SUBAPPLICATION logiBUS_AI_Calibrate_3P_IDA_OPC (* logiBUS_AI_IDA (Analog-Eingang) mit 3-Punkt-Kalibrierung (AR_CALIBRATE_3P_REF, unabhaengig gespeicherte Rohwerte X_MIN/X_MID/X_MAX + Referenzwerte MIN_REF/MID_REF/MAX_REF alle INI-persistiert) auf VT-Zahlenfelder (Rohwert + kalibrierter Wert, je eigene CNumberVariable) + Bargraph (kalibriert) + 3 VT-Tasten (C_MIN/C_MID/C_MAX) + OPC-UA (Rohwert DWORD + kalibrierter Wert REAL, generisch, ein Kanal). Fuer Sensoren mit definierter Mittelstellung (z.B. Lenkwinkelsensor: links/geradeaus/rechts) statt reiner 2-Punkt-Linearisierung. *)
  (* Standard: 61499-2; Description: Copyright (c) 2026 Meisterschulen am Ostbahnhof This program and the accompanying materials are made available under the terms of the Eclipse Public License 2.0 which is available at https://www.eclipse.org/legal/epl-2.0/ SPDX-License-Identifier: EPL-2.0 *)
  (* Version 1.2, 2026-09-18, Franz Höpfinger, Meisterschulen am Ostbahnhof, AR_CALIBRATE_3P_REF.C_MIN/C_MID/C_MAX von AX-Sockets auf reine EventInputs umgestellt (Franz-Entscheidung, siehe AR_CALIBRATE_2P_REF) - AX_BOOL_TO_X_MIN/_MID/_MAX entfallen ersatzlos, die Merge-Ketten verbinden jetzt direkt per EventConnection mit CALIBRATE.C_MIN/C_MID/C_MAX. *)
  (* Version 1.3, 2026-09-18, Franz Höpfinger, Meisterschulen am Ostbahnhof, C_MIN/C_MAX-Merge-Ketten (2x E_MERGE_2 in Reihe) durch je einen E_MERGE_3 ersetzt, C_MID-Kette (3x E_MERGE_2) durch einen E_MERGE_4 - OR-Merge ist assoziativ, funktional identisch. Siehe logiBUS_AI_Calibrate_IDA_OPC v1.4. *)
  (* Version 1.4, 2026-09-18, Franz Höpfinger, Meisterschulen am Ostbahnhof, Franz: 'kann eine SUB sein' - logiBUS_AI_IDA+AD_SPLIT_2+AD_PUBLISH_RAW+AD_TO_AUDI+AUDI_SPLIT_2+Q_NumericValue_RAW+AUDI_TO_AR durch neue SubApp logiBUS_AI_Raw_VT_AR_OPC ersetzt, AR_SPLIT_2+AR_PUBLISH_CAL+Q_NumericValue_CAL durch die bereits bestehende SubApp AR_TO_Q_Publish_OPC (dort um optionales INITO ergaenzt) - identisch zu logiBUS_AI_Calibrate_IDA_OPC v1.6. Die AX_SUBSCRIBE_MIN-Init-Kette haengt jetzt an PublishCal.INITO statt AR_PUBLISH_CAL.INITO; die vorherige Verkettung AD_PUBLISH_RAW.INITO->AR_PUBLISH_CAL.INIT entfaellt (beide Publishes sind voneinander unabhaengig, initialisieren jetzt unabhaengig/auto). *)
  (* Version 1.5, 2026-09-18, Franz Höpfinger, Meisterschulen am Ostbahnhof, Franz: 'genau so umbauen wie den anderen' (logiBUS_AI_Calibrate_IDA_OPC) - NUR fuer C_MIN/C_MAX: AX_SUBSCRIBE_MIN/MAX + AX_RF_TRIG_MIN/MAX (Toggle-Subscribe, ID_MIN_READ/ID_MAX_READ, beide ueberall unbenutzt) ersatzlos entfernt, ersetzt durch je eine Button_Method_IE (TriggerMIN/TriggerMAX) mit neuer Methodenadresse ID_MIN_METHOD/ID_MAX_METHOD. C_MID BEWUSST NICHT umgestellt: Fahrwerk_Mittelpunkt_Automatik.SUB (Achslenkung, STG1) triggert C_MID lokal (selbe Station!) ueber genau diesen Toggle-Kanal (ID_MID_READ), weil lokaler CALL_METHOD auf derselben Station laut 4diac-Doku nicht funktioniert (FORTE-Log: 'Cannot perform action CALL_METHOD locally') - siehe Fahrwerk_Mittelpunkt_Automatik.SUB v2.2/BERICHT_2026-09-16 Abschnitt 13-15. AX_SUBSCRIBE_MID/AX_RF_TRIG_MID/SERVER_MID_TRIGGER/E_MERGE_MID (E_MERGE_4) bleiben daher unveraendert bestehen. Die OPC_UA_VERNETZUNG.md Punkt 14-Regel (kein Event-Pegel-Event-Umweg) gilt nur fuer echte CROSS-STATION-Trigger, nicht fuer diesen Sonderfall auf derselben Station. *)
  (* Version 1.6, 2026-09-18, Franz Höpfinger, Meisterschulen am Ostbahnhof, Franz: 'TriggerMIN TriggerMAX bitte TriggerMID genau gleich machen' - Button_C_MID + SERVER_MID_TRIGGER (Button/Methode-Teil) durch eine SubApp TriggerMID (Button_Method_IE) ersetzt, strukturell identisch zu TriggerMIN/TriggerMAX. Der lokale Toggle-Kanal (AX_SUBSCRIBE_MID+AX_RF_TRIG_MID) bleibt bestehen (siehe v1.5-Begruendung), wird aber jetzt sauber getrennt als zusaetzliche Quelle in E_MERGE_MID gemergt (E_MERGE_4 -> E_MERGE_3: TriggerMID.IND + AX_RF_TRIG_MID.ER/EF) statt als 4. Quelle in einem grossen Merge mit SERVER_0 direkt inline verdrahtet zu sein. *)
  (* Version 1.7, 2026-09-18, Franz Höpfinger, Meisterschulen am Ostbahnhof, Franz: 'MID, MIN und MAX sind GLEICH' - AX_SUBSCRIBE_MID/AX_RF_TRIG_MID/E_MERGE_MID (der lokale Toggle-Kanal aus v1.5/v1.6) ersatzlos entfernt, ID_MID_READ entfaellt. TriggerMID ist jetzt eine reine Button_Method_IE-Instanz, 1:1 baugleich zu TriggerMIN/TriggerMAX, direkt auf CALIBRATE.C_MID verdrahtet. ACHTUNG: Fahrwerk_Mittelpunkt_Automatik.SUB (Achslenkung/Hangausgleich) toggelt/publiziert weiterhin auf den bisherigen ID_MID_TRIGGER_WRITE-Knoten, den jetzt niemand mehr abonniert - dieser Pfad ist damit funktionslos, bis Fahrwerk_Mittelpunkt_Automatik.SUB auf einen Aufruf von ID_MID_TRIGGER_METHOD umgestellt wird (lokaler CALL_METHOD schlug bisher fehl, siehe v1.5 - noch ungeklaert, wie das dort geloest wird). *)
  (* Version 1.1, 2026-09-11, Franz Höpfinger, Meisterschulen am Ostbahnhof, C_MID zusaetzlich per lokalem SERVER_0-Methodenaufruf (ID_MID_TRIGGER_METHOD, ACTION=CREATE_METHOD) ausloesbar - reiner RPC-Trigger fuer lokale Aufrufer (z.B. Achslenkung_Automatik.SUB per CLIENT_0), kein Toggle/PUBLISH/SUBSCRIBE-Umweg noetig wie beim echten Remote-Web-Kanal (ID_MID_READ). Per E_MERGE_MID_C mit dem bestehenden Button/Web-Merge zusammengefuehrt. *)
  (* Version 1.0, 2026-09-11, Franz Höpfinger, Meisterschulen am Ostbahnhof, 3-Punkt-Pendant zu logiBUS_AI_Calibrate_IDA_OPC (AR_CALIBRATE_3P_REF statt AR_CALIBRATE_2P_REF, 3 statt 2 Kalibrierpunkte/Tasten/Referenzwerte) - Sample fuer Sensoren mit Mittelstellung, siehe Workspace_AI_Calibrate_3P. *)
  (* Version 1.8, 2026-09-20, Franz Höpfinger, Meisterschulen am Ostbahnhof, Rohwert-Anzeige an den 3 Kalibrierpunkten (Min/Mid/Max-Raw) ergaenzt, analog zu logiBUS_AI_Calibrate_IDA_OPC v1.7 (Franz: 'im Web-Panel und im IOP die Roh-Werte mit anzeigen'). CALIBRATE.X_MIN/X_MID/X_MAX (AR2, bisher nur an INI_X_MIN/INI_X_MID/INI_X_MAX angeschlossen) werden ueber neue TapMinRaw/TapMidRaw/TapMaxRaw (MyLib::sys::AR2_TAP_TO_AR) abgezapft, ohne die bestehende Persistenz-/Restore-Kette zu aendern, und ueber neue PublishMinRaw/PublishMidRaw/PublishMaxRaw (MyLib::sys::AR_TO_Q_Publish_OPC) als reine Nur-Lese-Anzeige (VT CNumberVariable + OPC-UA Publish) exponiert. Neue InputVars stObjMinRaw/stObjMidRaw/stObjMaxRaw (VT-Objekt) + ID_MIN_RAW_WRITE/ID_MID_RAW_WRITE/ID_MAX_RAW_WRITE (OPC-UA-Adresse). *)
  (* Version 1.10, 2026-09-21, Franz Höpfinger, Meisterschulen am Ostbahnhof, Code-Review-Fund (PR #260): INI_X_MID/INI_X_MAX.DEFAULT_VALUE standen auf REAL#0.5/1.0 statt 0.0 - AR_CALIBRATE_3P_REF's neue xMidCal/xMaxCal-Kalibriert-Flags (v1.3, pruefen X_MID.DI1/X_MAX.DI1 <> 0.0) latchten dadurch bei JEDEM Boot sofort TRUE, obwohl MID/MAX nie kalibriert wurden (fabricated references statt Partial-Kalibrierung-Fallback). Defaults auf REAL#0.0 korrigiert, passend zu INI_X_MIN und zum Flag-Vergleich. *)
  (* Version 1.9, 2026-09-21, Franz Höpfinger, Meisterschulen am Ostbahnhof, AR_CALIBRATE_3P_REF hat jetzt ein INIT/QI/QO-Enable-Pattern (Bugfix MIN-vor-MID + xClipping) - CALIBRATE bekommt Parameter QI=TRUE (wie die INI_X_MIN/X_MID/X_MAX-Instanzen), sonst bleibt die FB im START-Zustand haengen und REQ laeuft nie. *)
  (* Version 1.11, 2026-09-26, Franz Höpfinger, Meisterschulen am Ostbahnhof, INI_MID_REF.DEFAULT_VALUE stand auf REAL#50.0 statt 0.0 - passte nicht zur dokumentierten Kalibrierwert-Konvention (-100=Links-Anschlag/0=Mitte/+100=Rechts-Anschlag, siehe ACHSLENKUNG_WINKEL_CAL_LOC_WRITE-Kommentar in SubStrings_STG1.gcf). Bei Achslenkung Winkel B02 entdeckt/bestaetigt (Franz), korrigiert auf REAL#0.0, passend zu INI_MIN_REF/INI_MAX_REF's Vorzeichen-Konvention. *)
  PACKAGE MyLib::sys;
  IMPORT isobus::UT::Q::const::IDs::ID_NULL;
  IMPORT logiBUS::io::AI::logiBUS_AI;
  IMPORT logiBUS::io::AI::logiBUS_AI_S;
  IMPORT logiBUS::utils::conversion::phys::NumericObjectPool_S;
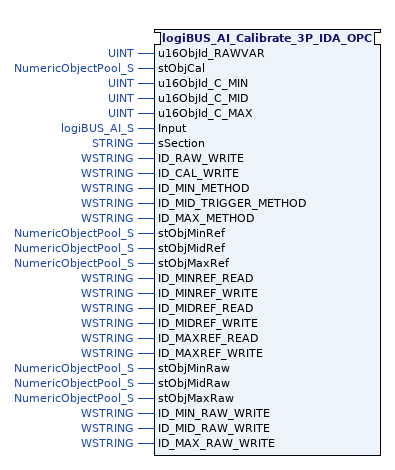
  VAR_INPUT
    u16ObjId_RAWVAR : UINT := ID_NULL; (* Object ID CNumberVariable (Rohwert 0-4095, unkalibriert, reine Diagnose-Anzeige) *)
    stObjCal : logiBUS::utils::conversion::phys::NumericObjectPool_S := (u16ObjId := ID_NULL, r32Scale := 1.0, i32Offset := 0, u8Decimals := 1); (* Object ID + Scale/Offset/Decimals CNumberVariable (kalibrierter Wert, eigene, unabhaengige CNumberVariable) *)
    u16ObjId_C_MIN : UINT := ID_NULL; (* Object ID Taste 'C_MIN' (Min-Position anfahren, dann druecken) *)
    u16ObjId_C_MID : UINT := ID_NULL; (* Object ID Taste 'C_MID' (Mittelstellung anfahren, dann druecken) *)
    u16ObjId_C_MAX : UINT := ID_NULL; (* Object ID Taste 'C_MAX' (Max-Position anfahren, dann druecken) *)
    Input : logiBUS::io::AI::logiBUS_AI_S := logiBUS_AI::Invalid; (* Identify the Input AnalogInput_I1..I8 *)
    sSection : STRING; (* INI-Sektionsname fuer X_MIN/X_MID/X_MAX/MIN_REF/MID_REF/MAX_REF-Persistenz - pro Kanal eindeutig, sonst kollidieren die Kanaele in settings.ini *)
    ID_RAW_WRITE : WSTRING; (* Rohwert-Ruckmelde-Adresse (DWORD 0-4095, ACTION=PUBLISH) *)
    ID_CAL_WRITE : WSTRING; (* Kalibrierter-Wert-Ruckmelde-Adresse (REAL, ACTION=PUBLISH) *)
    ID_MIN_METHOD : WSTRING; (* Methodenadresse (ACTION=CREATE_METHOD) fuer den argumentlosen C_MIN-Trigger - gleichberechtigt zur lokalen VT-Taste aufrufbar, sowohl vom OPC-UA-Dashboard als auch per CLIENT_0 von einer anderen Station (siehe OPC_UA_VERNETZUNG.md Punkt 14 - kein Toggle/Subscribe-Umweg mehr) *)
    ID_MID_TRIGGER_METHOD : WSTRING; (* Methodenadresse (ACTION=CREATE_METHOD) fuer den argumentlosen C_MID-Trigger - siehe ID_MIN_METHOD *)
    ID_MAX_METHOD : WSTRING; (* Methodenadresse (ACTION=CREATE_METHOD) fuer den argumentlosen C_MAX-Trigger - siehe ID_MIN_METHOD *)
    stObjMinRef : logiBUS::utils::conversion::phys::NumericObjectPool_S := (u16ObjId := ID_NULL, r32Scale := 1.0, i32Offset := 0, u8Decimals := 1); (* Object ID + Scale/Offset/Decimals CNumberVariable (MIN_REF-Referenzwert, VT-Eingabefeld + OPC-UA) *)
    stObjMidRef : logiBUS::utils::conversion::phys::NumericObjectPool_S := (u16ObjId := ID_NULL, r32Scale := 1.0, i32Offset := 0, u8Decimals := 1); (* Object ID + Scale/Offset/Decimals CNumberVariable (MID_REF-Referenzwert, VT-Eingabefeld + OPC-UA) *)
    stObjMaxRef : logiBUS::utils::conversion::phys::NumericObjectPool_S := (u16ObjId := ID_NULL, r32Scale := 1.0, i32Offset := 0, u8Decimals := 1); (* Object ID + Scale/Offset/Decimals CNumberVariable (MAX_REF-Referenzwert, VT-Eingabefeld + OPC-UA) *)
    ID_MINREF_READ : WSTRING; (* Remote-Subscribe-Adresse MIN_REF-Referenzwert (REAL, ACTION=SUBSCRIBE) *)
    ID_MINREF_WRITE : WSTRING; (* Remote-Echo-Adresse MIN_REF-Referenzwert (REAL, ACTION=PUBLISH) *)
    ID_MIDREF_READ : WSTRING; (* Remote-Subscribe-Adresse MID_REF-Referenzwert (REAL, ACTION=SUBSCRIBE) *)
    ID_MIDREF_WRITE : WSTRING; (* Remote-Echo-Adresse MID_REF-Referenzwert (REAL, ACTION=PUBLISH) *)
    ID_MAXREF_READ : WSTRING; (* Remote-Subscribe-Adresse MAX_REF-Referenzwert (REAL, ACTION=SUBSCRIBE) *)
    ID_MAXREF_WRITE : WSTRING; (* Remote-Echo-Adresse MAX_REF-Referenzwert (REAL, ACTION=PUBLISH) *)
    stObjMinRaw : logiBUS::utils::conversion::phys::NumericObjectPool_S := (u16ObjId := ID_NULL, r32Scale := 1.0, i32Offset := 0, u8Decimals := 1); (* Object ID + Scale/Offset/Decimals CNumberVariable (Rohwert am MIN-Kalibrierpunkt, reine Diagnose-Anzeige) *)
    stObjMidRaw : logiBUS::utils::conversion::phys::NumericObjectPool_S := (u16ObjId := ID_NULL, r32Scale := 1.0, i32Offset := 0, u8Decimals := 1); (* Object ID + Scale/Offset/Decimals CNumberVariable (Rohwert am MID-Kalibrierpunkt, reine Diagnose-Anzeige) *)
    stObjMaxRaw : logiBUS::utils::conversion::phys::NumericObjectPool_S := (u16ObjId := ID_NULL, r32Scale := 1.0, i32Offset := 0, u8Decimals := 1); (* Object ID + Scale/Offset/Decimals CNumberVariable (Rohwert am MAX-Kalibrierpunkt, reine Diagnose-Anzeige) *)
    ID_MIN_RAW_WRITE : WSTRING; (* Rohwert-am-MIN-Kalibrierpunkt-Publish-Adresse (REAL, ACTION=PUBLISH) *)
    ID_MID_RAW_WRITE : WSTRING; (* Rohwert-am-MID-Kalibrierpunkt-Publish-Adresse (REAL, ACTION=PUBLISH) *)
    ID_MAX_RAW_WRITE : WSTRING; (* Rohwert-am-MAX-Kalibrierpunkt-Publish-Adresse (REAL, ACTION=PUBLISH) *)
  END_VAR
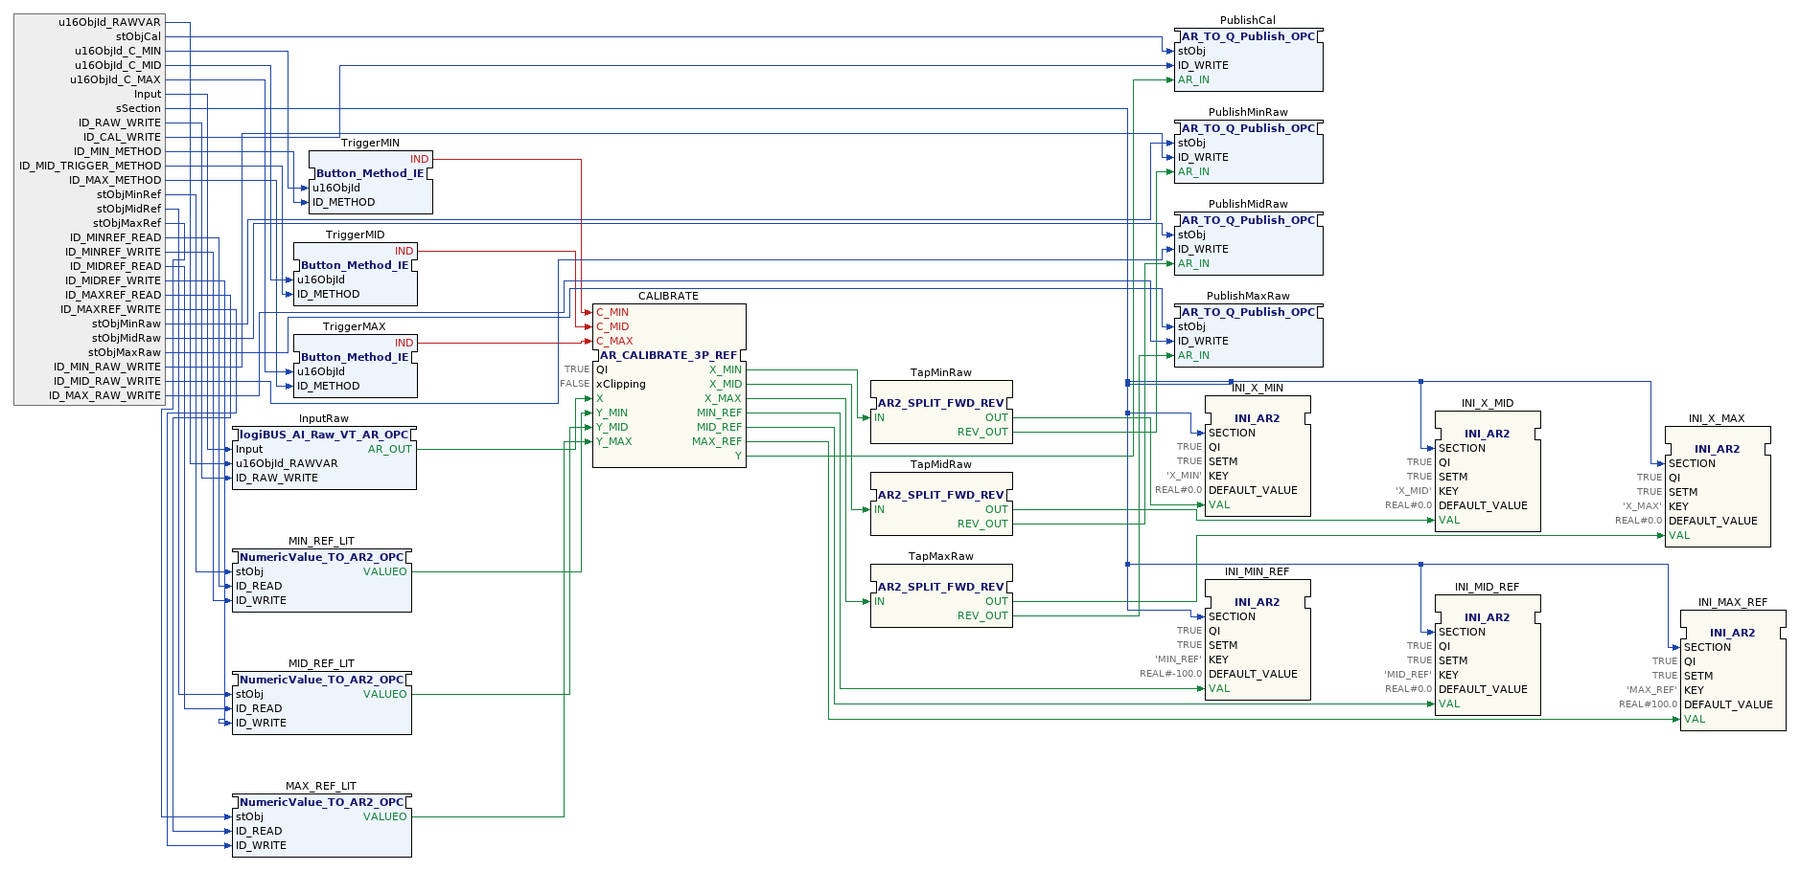
  FBS
    CALIBRATE : adapter::Engineering::measurements::AR_CALIBRATE_3P_REF(QI := TRUE, xClipping := FALSE);
    INI_X_MIN : eclipse4diac::storage::INI_AR2(QI := TRUE, SETM := TRUE, KEY := 'X_MIN', DEFAULT_VALUE := REAL#0.0);
    INI_X_MID : eclipse4diac::storage::INI_AR2(QI := TRUE, SETM := TRUE, KEY := 'X_MID', DEFAULT_VALUE := REAL#0.0);
    INI_X_MAX : eclipse4diac::storage::INI_AR2(QI := TRUE, SETM := TRUE, KEY := 'X_MAX', DEFAULT_VALUE := REAL#0.0);
    INI_MIN_REF : eclipse4diac::storage::INI_AR2(QI := TRUE, SETM := TRUE, KEY := 'MIN_REF', DEFAULT_VALUE := REAL#-100.0);
    INI_MID_REF : eclipse4diac::storage::INI_AR2(QI := TRUE, SETM := TRUE, KEY := 'MID_REF', DEFAULT_VALUE := REAL#0.0);
    INI_MAX_REF : eclipse4diac::storage::INI_AR2(QI := TRUE, SETM := TRUE, KEY := 'MAX_REF', DEFAULT_VALUE := REAL#100.0);
    TapMinRaw : adapter::events::bidirectional::AR2_SPLIT_FWD_REV;
    TapMidRaw : adapter::events::bidirectional::AR2_SPLIT_FWD_REV;
    TapMaxRaw : adapter::events::bidirectional::AR2_SPLIT_FWD_REV;
  END_FBS
  SUBAPPS
    InputRaw : MyLib::sys::logiBUS_AI_Raw_VT_AR_OPC;
    MIN_REF_LIT : MyLib::sys::NumericValue_TO_AR2_OPC;
    MID_REF_LIT : MyLib::sys::NumericValue_TO_AR2_OPC;
    MAX_REF_LIT : MyLib::sys::NumericValue_TO_AR2_OPC;
    TriggerMIN : MyLib::sys::Button_Method_IE;
    TriggerMID : MyLib::sys::Button_Method_IE;
    TriggerMAX : MyLib::sys::Button_Method_IE;
    PublishCal : MyLib::sys::AR_TO_Q_Publish_OPC;
    PublishMinRaw : MyLib::sys::AR_TO_Q_Publish_OPC;
    PublishMidRaw : MyLib::sys::AR_TO_Q_Publish_OPC;
    PublishMaxRaw : MyLib::sys::AR_TO_Q_Publish_OPC;
  END_SUBAPPS
  EVENT_CONNECTIONS
    TriggerMIN.IND TO CALIBRATE.C_MIN;
    TriggerMID.IND TO CALIBRATE.C_MID;
    TriggerMAX.IND TO CALIBRATE.C_MAX;
  END_CONNECTIONS
  DATA_CONNECTIONS
    Input TO InputRaw.Input;
    u16ObjId_RAWVAR TO InputRaw.u16ObjId_RAWVAR;
    stObjCal TO PublishCal.stObj;
    u16ObjId_C_MIN TO TriggerMIN.u16ObjId;
    u16ObjId_C_MID TO TriggerMID.u16ObjId;
    u16ObjId_C_MAX TO TriggerMAX.u16ObjId;
    sSection TO INI_X_MIN.SECTION;
    sSection TO INI_X_MID.SECTION;
    sSection TO INI_X_MAX.SECTION;
    sSection TO INI_MIN_REF.SECTION;
    sSection TO INI_MID_REF.SECTION;
    sSection TO INI_MAX_REF.SECTION;
    ID_RAW_WRITE TO InputRaw.ID_RAW_WRITE;
    ID_CAL_WRITE TO PublishCal.ID_WRITE;
    ID_MIN_METHOD TO TriggerMIN.ID_METHOD;
    ID_MID_TRIGGER_METHOD TO TriggerMID.ID_METHOD;
    ID_MAX_METHOD TO TriggerMAX.ID_METHOD;
    stObjMinRef TO MIN_REF_LIT.stObj;
    ID_MINREF_READ TO MIN_REF_LIT.ID_READ;
    ID_MINREF_WRITE TO MIN_REF_LIT.ID_WRITE;
    stObjMidRef TO MID_REF_LIT.stObj;
    ID_MIDREF_READ TO MID_REF_LIT.ID_READ;
    ID_MIDREF_WRITE TO MID_REF_LIT.ID_WRITE;
    stObjMaxRef TO MAX_REF_LIT.stObj;
    ID_MAXREF_READ TO MAX_REF_LIT.ID_READ;
    ID_MAXREF_WRITE TO MAX_REF_LIT.ID_WRITE;
    stObjMinRaw TO PublishMinRaw.stObj;
    ID_MIN_RAW_WRITE TO PublishMinRaw.ID_WRITE;
    stObjMidRaw TO PublishMidRaw.stObj;
    ID_MID_RAW_WRITE TO PublishMidRaw.ID_WRITE;
    stObjMaxRaw TO PublishMaxRaw.stObj;
    ID_MAX_RAW_WRITE TO PublishMaxRaw.ID_WRITE;
  END_CONNECTIONS
  ADAPTER_CONNECTIONS
    InputRaw.AR_OUT TO CALIBRATE.X;
    CALIBRATE.X_MIN TO TapMinRaw.IN;
    TapMinRaw.OUT TO INI_X_MIN.VAL;
    TapMinRaw.REV_OUT TO PublishMinRaw.AR_IN;
    CALIBRATE.X_MID TO TapMidRaw.IN;
    TapMidRaw.OUT TO INI_X_MID.VAL;
    TapMidRaw.REV_OUT TO PublishMidRaw.AR_IN;
    CALIBRATE.X_MAX TO TapMaxRaw.IN;
    TapMaxRaw.OUT TO INI_X_MAX.VAL;
    TapMaxRaw.REV_OUT TO PublishMaxRaw.AR_IN;
    CALIBRATE.MIN_REF TO INI_MIN_REF.VAL;
    CALIBRATE.MID_REF TO INI_MID_REF.VAL;
    CALIBRATE.MAX_REF TO INI_MAX_REF.VAL;
    MIN_REF_LIT.VALUEO TO CALIBRATE.Y_MIN;
    MID_REF_LIT.VALUEO TO CALIBRATE.Y_MID;
    MAX_REF_LIT.VALUEO TO CALIBRATE.Y_MAX;
    CALIBRATE.Y TO PublishCal.AR_IN;
  END_CONNECTIONS
END_SUBAPPLICATION
